FUNCTION_BLOCK AE_CLIENT_0 (* Trigger a remote OPC-UA method call via CLIENT_0, driven by an AE adapter Socket (1 Event) *)
  (* Standard: 61499-2; Description: Copyright (c) 2026 HR Agrartechnik GmbH This program and the accompanying materials are made available under the terms of the Eclipse Public License 2.0 which is available at https://www.eclipse.org/legal/epl-2.0/ SPDX-License-Identifier: EPL-2.0 *)
  (* Version 1.0, 2026-09-03, Franz Höpfinger, HR Agrartechnik GmbH, initial API and implementation and/or initial documentation *)
  PACKAGE adapter::net;
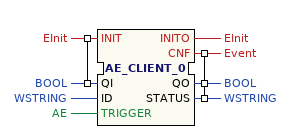
  EVENT_INPUT
    INIT : EInit WITH QI; (* Initialization *)
  END_EVENT
  EVENT_OUTPUT
    INITO : EInit; (* Initialization Confirm *)
    CNF WITH QO, STATUS; (* QO/STATUS updated *)
  END_EVENT
  VAR_INPUT
    QI : BOOL;
    ID : WSTRING;
  END_VAR
  VAR_OUTPUT
    QO : BOOL; (* QO von CLIENT_0_1 *)
    STATUS : WSTRING; (* STATUS von CLIENT_0_1 *)
  END_VAR
  SOCKETS
    TRIGGER : adapter::types::unidirectional::AE; (* Trigger *)
  END_SOCKETS
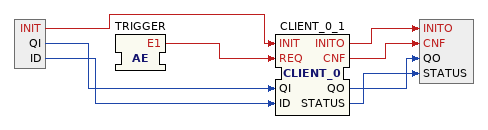
  FBS
    CLIENT_0_1 : iec61499::net::CLIENT_0;
  END_FBS
  EVENT_CONNECTIONS
    INIT TO CLIENT_0_1.INIT;
    CLIENT_0_1.INITO TO INITO;
    TRIGGER.E1 TO CLIENT_0_1.REQ;
    CLIENT_0_1.CNF TO CNF;
  END_CONNECTIONS
  DATA_CONNECTIONS
    QI TO CLIENT_0_1.QI;
    ID TO CLIENT_0_1.ID;
    CLIENT_0_1.QO TO QO;
    CLIENT_0_1.STATUS TO STATUS;
  END_CONNECTIONS
END_FUNCTION_BLOCK
